FUNCTION_BLOCK ADSLogger IMPLEMENTS EventLogger
VAR_INPUT
END_VAR
VAR_OUTPUT
END_VAR
VAR
  _level: EventLevel;
  _disable_ads_output: BOOL;
  _mask: DWORD;
  _prefix: STRING(15);
  _formatted_output: STRING(255);
END_VAR

METHOD PRIVATE ads_log
VAR_INPUT
  ev: EventMessage;
END_VAR
VAR
END_VAR
mask := create_mask(ev.level);
prefix := create_prefix(ev.level);

formatted_output := CONCAT(prefix, ev.message);

IF NOT disable_ads_output THEN
  ADSLOGSTR(mask, formatted_output, '');
END_IF
END_METHOD

METHOD PRIVATE create_mask : DWORD
VAR_INPUT
  level: EventLevel;
END_VAR
CASE level OF
EventLevel.INFO:
  create_mask := ADSLOG_MSGTYPE_HINT;
EventLevel.WARNING:
  create_mask := ADSLOG_MSGTYPE_WARN;
EventLevel.ERROR:
  create_mask := ADSLOG_MSGTYPE_ERROR;
ELSE
  create_mask := ADSLOG_MSGTYPE_HINT;
END_CASE
END_METHOD

METHOD PRIVATE create_prefix : STRING(15)
VAR_INPUT
  level: EventLevel;
END_VAR
CASE level OF
EventLevel.INFO:
  create_prefix := ' | Info: ';
EventLevel.WARNING:
  create_prefix := ' | Warning: ';
EventLevel.ERROR:
  create_prefix := ' | Error: ';
ELSE
  create_prefix := ' | Undefined: ';
END_CASE
END_METHOD

PROPERTY INTERNAL disable_ads_output : BOOL
GET
disable_ads_output := _disable_ads_output;
END_GET
SET
_disable_ads_output := disable_ads_output;
END_SET
END_PROPERTY

PROPERTY INTERNAL formatted_output : STRING(255)
GET
formatted_output := _formatted_output;
END_GET
SET // PRIVATE
_formatted_output := formatted_output;
END_SET
END_PROPERTY

PROPERTY PUBLIC level : EventLevel
GET
level := _level;
END_GET
SET
_level := level;
END_SET
END_PROPERTY

PROPERTY INTERNAL mask : DWORD
GET
mask := _mask;
END_GET
SET // PRIVATE
_mask := mask;
END_SET
END_PROPERTY

PROPERTY INTERNAL prefix : STRING(15)
GET
prefix := _prefix;
END_GET
SET // PRIVATE
_prefix := prefix;
END_SET
END_PROPERTY

METHOD PUBLIC submit_event_message
VAR_INPUT
	ev: EventMessage;
END_VAR
IF ev.level >= level THEN
  ads_log(ev);
END_IF
END_METHOD

END_FUNCTION_BLOCK

(* stored: Version 1.1.0.1, ProductVersion 3.1.4024.9
   POU ADSLogger: Id {f353a23b-59c1-4eb7-b1b3-77f5986ff606}, SpecialFunc None
   Method ads_log: Id {1bc6e817-4323-49bf-a63f-a94d3b6c886f}
   Method create_mask: Id {aee6a054-3e4f-421c-aca5-2c735f9fea76}
   Method create_prefix: Id {e6393b63-a206-438e-accf-a721f61f3d0a}
   Property disable_ads_output: Id {7e9c1897-64d5-455a-b20b-e82b4706fc80}
   Get Get: Id {249061bd-6c70-46d6-a135-7e502181640a}
   Set Set: Id {41f678c7-9359-4213-abb0-e87b5beeefc5}
   Property formatted_output: Id {c00d9c99-7aed-49b0-83c9-9c5fba96f988}
   Get Get: Id {cb587932-271f-416f-b6a0-4af026f4953f}
   Set Set: Id {8bc1fa17-0d69-4124-b2c4-148f2b65324b}
   Property level: Id {a8405867-ed20-4229-ac83-fd765a22d2e1}
   Get Get: Id {e4dc5a89-34cc-4104-955c-43c82263873f}
   Set Set: Id {0a7594a5-f4cb-4c89-8bae-3f536563dccb}
   Property mask: Id {494ef503-2861-4c0f-84f8-541fba4f652f}
   Get Get: Id {a0b8587b-6cb6-4514-8d0b-783e5f031085}
   Set Set: Id {c49ea54b-51ab-4a9a-b5b0-f3313dcf06e5}
   Property prefix: Id {323f41d0-a33a-4170-aaca-6778f0d96f7d}
   Get Get: Id {8ee79c6b-0c1f-4ac5-bc2d-f4f7faabd841}
   Set Set: Id {d2420567-3b92-48d5-8816-decae5ecdad9}
   Method submit_event_message: Id {72fa51cd-5f83-427b-a2c1-e007bce7d269} *)
